FUNCTION_BLOCK FB_IODEV_CH_ANLG_OUT EXTENDS FB_IODEV_CH_ANALOG
VAR_INPUT
END_VAR
VAR_OUTPUT
END_VAR
VAR
	// Physical active output signal.
	// Read-Only access via OPC UA.
	{attribute 'OPC.UA.DA' := '1'}
	{attribute 'OPC.UA.DA.Access' := '1'}
	q_nValue	AT %Q*:	INT;

	// Output values
	// Configured for R/W OPC UA Data Access !!!
	{attribute 'OPC.UA.DA' := '1'}
	{attribute 'OPC.UA.DA.Access' := '3'}
	nValue:			INT;	// Computed output value
	{attribute 'OPC.UA.DA' := '1'}
	{attribute 'OPC.UA.DA.Access' := '3'}
	lrValueUser:	LREAL;	// Output value in User Units
	
END_VAR

METHOD M_Compute
VAR_INPUT
END_VAR
//
// For CONVERSION_IODEV_NONE nValue is used for output.
// In this case nValue is copied into lrValueUser.
// For others nValue is calculated from the User value.
//
CASE nConversion OF
	CONVERSION_IODEV_NONE:
		lrValueUser := INT_TO_LREAL(nValue);	// Copy nValue into lrValueUser
	CONVERSION_IODEV_LINEAR:
		nValue	:= LREAL_TO_INT(lrPar1 * lrValueUser  +  lrPar2);
	CONVERSION_IODEV_QUADRATIC:
		nValue	:= LREAL_TO_INT(lrPar1 * lrValueUser * lrValueUser  +  lrPar2 * lrValueUser  +  lrPar3);
	CONVERSION_IODEV_EXP:
		nValue	:= LREAL_TO_INT(EXP (lrPar1 * lrValueUser  +  lrPar2));
	CONVERSION_IODEV_EXP10:
		nValue	:= LREAL_TO_INT(EXPT (10.0, (lrPar1 * lrValueUser  +  lrPar2)));
END_CASE

// Set the output
q_nValue	:= nValue;
END_METHOD

METHOD M_Configure
VAR_INPUT
END_VAR
VAR_INPUT
	in_eConversion:	E_IODEV_CONVERSION;
	in_lrPar1:		LREAL := 0.0;
	in_lrPar2:		LREAL := 0.0;
	in_lrPar3:		LREAL := 0.0;
END_VAR
nConversion		:= in_eConversion;
lrPar1			:= in_lrPar1;
lrPar2			:= in_lrPar2;
lrPar3			:= in_lrPar3;

// Set output to zero
q_nValue		:= 0;
nValue			:= 0;
lrValueUser		:= 0.0;
END_METHOD

METHOD M_Reset
VAR_INPUT
END_VAR
nConversion	:= CONVERSION_IODEV_NONE;
lrPar1			:= 0.0;
lrPar2			:= 0.0;
lrPar3			:= 0.0;

// Set output to zero
q_nValue		:= 0;
nValue			:= 0;
lrValueUser		:= 0.0;
END_METHOD

END_FUNCTION_BLOCK

(* stored: Version 1.1.0.1, ProductVersion 3.1.4024.12
   POU FB_IODEV_CH_ANLG_OUT: Id {67f95494-b3e4-4f98-a441-ae06b4bfb7ea}, SpecialFunc None
   Method M_Compute: Id {993282a3-6fda-4906-af79-abdfd6b3bb4c}
   Method M_Configure: Id {b81cbc58-5541-48b1-98c2-0e37caff6f05}
   Method M_Reset: Id {fe03e4f6-18aa-4416-8d34-0fbc6e36d5e8} *)
